// SIMATIC S7-200 project (STEP 7-Micro/WIN), CPU 224 REL 02.01

SYMBOL_TABLE USUARIO1
TARJETERO        I0.0
CELULA           I0.1
FC_SUBIDA        I0.2
FC_BAJADA        I0.3
TERMICO          I0.5
M1_APERTURA      Q0.0
M1_CIERRE        Q0.1
END_SYMBOL_TABLE

ORGANIZATION_BLOCK PRINCIPAL:OB1
TITLE=COMENTARIOS DEL PROGRAMA
BEGIN
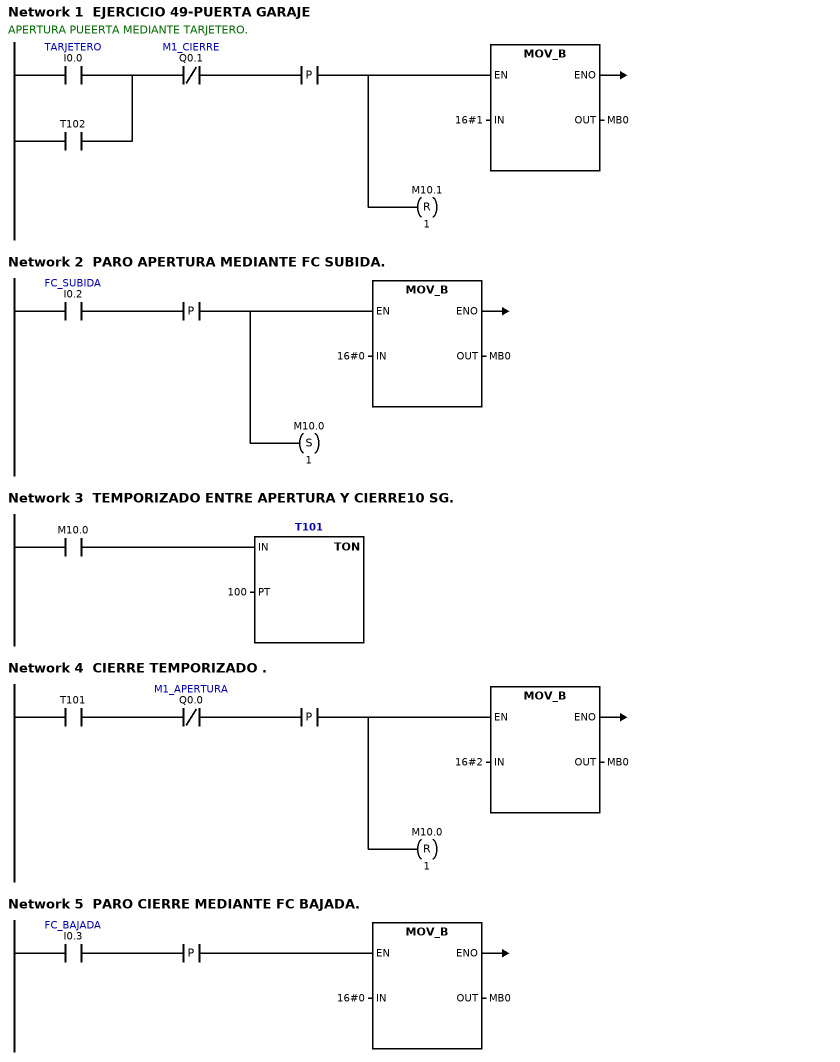
Network 1 // EJERCICIO 49-PUERTA GARAJE
// APERTURA PUEERTA MEDIANTE TARJETERO.
LD     TARJETERO:I0.0
O      T102
AN     M1_CIERRE:Q0.1
EU
MOVB   16#1, MB0
R      M10.1, 1
Network 2 // PARO APERTURA MEDIANTE FC SUBIDA.
LD     FC_SUBIDA:I0.2
EU
MOVB   16#0, MB0
S      M10.0, 1
Network 3 // TEMPORIZADO ENTRE APERTURA Y CIERRE10 SG.
LD     M10.0
TON    T101, 100
Network 4 // CIERRE TEMPORIZADO .
LD     T101
AN     M1_APERTURA:Q0.0
EU
MOVB   16#2, MB0
R      M10.0, 1
Network 5 // PARO CIERRE MEDIANTE FC BAJADA.
LD     FC_BAJADA:I0.3
EU
MOVB   16#0, MB0
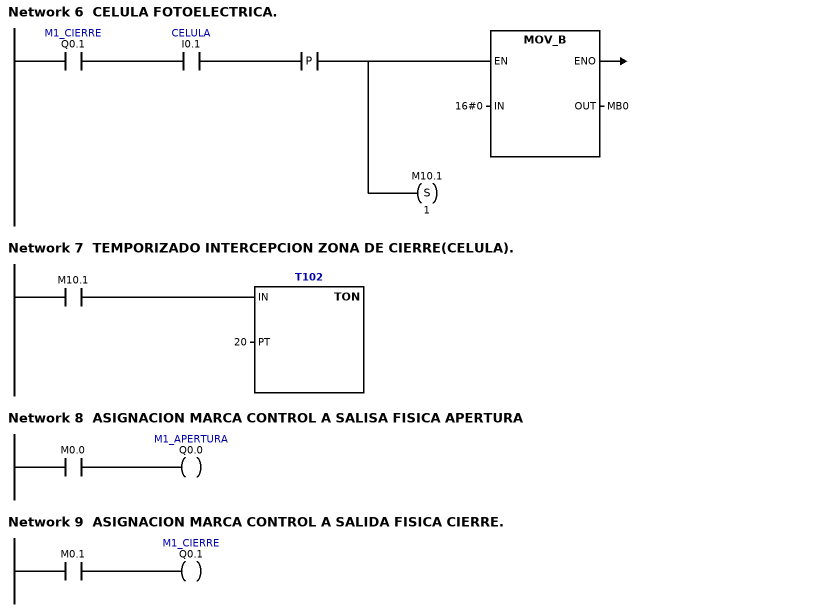
Network 6 // CELULA FOTOELECTRICA.
LD     M1_CIERRE:Q0.1
A      CELULA:I0.1
EU
MOVB   16#0, MB0
S      M10.1, 1
Network 7 // TEMPORIZADO INTERCEPCION ZONA DE CIERRE(CELULA).
LD     M10.1
TON    T102, 20
Network 8 // ASIGNACION MARCA CONTROL A SALISA FISICA APERTURA
LD     M0.0
=      M1_APERTURA:Q0.0
Network 9 // ASIGNACION MARCA CONTROL A SALIDA FISICA CIERRE.
LD     M0.1
=      M1_CIERRE:Q0.1
END_ORGANIZATION_BLOCK
